(* PLC project proyecto auto generado.project, CODESYS CODESYS V3.5 SP9 Patch 4 *)
(* stored: creationDateTime 2019-10-24T08:43:56.7165045, modificationDateTime 2019-10-17T10:33:55.5032294 *)

PROGRAM GEMMA

                    
                  
END_PROGRAM

PROGRAM A6

                    
                  
END_PROGRAM

PROGRAM A1

                    
                  
END_PROGRAM

PROGRAM A5

                    
                  
END_PROGRAM

PROGRAM A2

                    
                  
END_PROGRAM

PROGRAM F1

                    
                  
END_PROGRAM

PROGRAM F2

                    
                  
END_PROGRAM

PROGRAM F3

                    
                  
END_PROGRAM

PROGRAM F4

                    
                  
END_PROGRAM

PROGRAM F5

                    
                  
END_PROGRAM

PROGRAM D1

                    
                  
END_PROGRAM

PROGRAM D2

                    
                  
END_PROGRAM

PROGRAM D3

                    
                  
END_PROGRAM

CONFIGURATION Device Auto Generate
  RESOURCE Application ON PLC
    TASK MainTask(INTERVAL := T#20ms, PRIORITY := 1);
    PROGRAM GEMMA WITH MainTask : GEMMA;
  END_RESOURCE
END_CONFIGURATION
